FUNCTION_BLOCK FB_TransferLine EXTENDS StateMachine
VAR_INPUT
END_VAR
VAR_OUTPUT
END_VAR
VAR
	aBeltConveyors : ARRAY[1..2] OF FB_BeltConveyor;
	aRollerConveyors : ARRAY[1..3] OF FB_RollerConveyor;
	
	fbCounterSensor : FB_Sensor;
	fbPalletizer : FB_Palletizer;
	fbStepWorkerReady : FB_StepWorker;
	fbStepWorkerBusy : FB_StepWorker;
	
	fbChainController : FB_ChainController;
	
	scBeltConveyors : FB_BeltConveyors;
	scPostPalletizer : FB_PostPalletizer;
	scPrePalletizer : FB_PrePalletizer;
 
	fbTrig : R_TRIG;
	uiPackageCounter : UINT;
	i : UINT;
	bPackageOnTheWay : BOOL;
END_VAR

SUPER^();

FOR i := 1 TO 3 
DO
	IF i <> eTlMaxNumBeltConveyors
	THEN
		aBeltConveyors[i]();
	END_IF
	
	IF i <> eTlMaxNumRollerConveyors
	THEN
		aRollerConveyors[i]();
	END_IF
END_FOR

fbPalletizer();

METHOD PROTECTED   Busy : BOOL
VAR_INPUT
END_VAR
CASE fbStepWorkerBusy.uiStep OF

	eTlBusyStart: 
	
		//At start we check how many packages have passed the fbCounterSensor
		IF uiPackageCounter < 3
		THEN
		
			//activate the conveyors
			fbStepWorkerBusy.mNextStep(eTlStartEntranceConveyor);
			
		ELSIF uiPackageCounter = 3
		 AND NOT fbPalletizer.bAllPartsPresent
		THEN
 			//A package needs to reach the palletizer or a sensor is malfunctioning
			aBeltConveyors[eBeltConveyorEntrance].Off();
			fbStepWorkerBusy.mNextStep(eTlStartUpwardsConveyor);
		ELSIF uiPackageCounter = 3
		 AND fbPalletizer.bAllPartsPresent
	 	THEN
			//Execute the Palletizer
			aBeltConveyors[eBeltConveyorUpwards].Off();
			fbStepWorkerBusy.mNextStep(eTlExecutePalletizer);
		ELSIF uiPackageCounter > 3
		THEN
			//Error
		END_IF
		
	eTlStartEntranceConveyor:
		
		aBeltConveyors[eBeltConveyorEntrance].On();
		fbStepWorkerBusy.mAddCondition(fbCounterSensor.getSignal);
		fbStepWorkerBusy.mNextStep(eTlStartUpwardsConveyor);

	eTlStartUpwardsConveyor:
	
		aBeltConveyors[eBeltConveyorUpwards].On();
		fbStepWorkerBusy.mNextStep(eTlExecutePalletizer);
			 
	eTlExecutePalletizer:
		 
		fbPalletizer.Execute();
		fbStepWorkerBusy.mAddCondition(fbPalletizer.getDoneCycle);
		fbStepWorkerBusy.mNextStep(eTlBusyStart);
		 
	eTlSignalError:
	
		fbStepWorkerBusy.mNextStep(eTlBusyStart);
		Fault();	
		
		
END_CASE
END_METHOD

METHOD PROTECTED  Error : BOOL
VAR_INPUT
END_VAR
FOR i := 1 TO 3 
DO
	IF i <> eTlMaxNumBeltConveyors
	THEN
		aBeltConveyors[i].Off();
	END_IF
	
	IF i <> eTlMaxNumRollerConveyors
	THEN
		aRollerConveyors[i].Off();
	END_IF
END_FOR
END_METHOD

METHOD PROTECTED  Init : BOOL
VAR_INPUT
END_VAR
Start();
END_METHOD

METHOD PROTECTED  Ready : BOOL
VAR_INPUT
END_VAR
END_METHOD

END_FUNCTION_BLOCK

(* stored: Version 1.1.0.1, ProductVersion 3.1.4024.0
   POU FB_TransferLine: Id {2e7b366f-b9ef-4b13-bd70-7031bb32b800}, SpecialFunc None
   Method Busy: Id {3dde4417-0d0c-49da-9bd9-97065e9ed964}
   Method Error: Id {dcf9a9b3-729d-4763-8c13-3d1ffd1dfd1e}
   Method Init: Id {4357aa31-540d-408d-bbfa-5ee1874096be}
   Method Ready: Id {4f0f5542-23e8-48a2-84b3-069ccd15f633} *)
